VAR_GLOBAL
     g_xFirstPass: BOOL := TRUE;
    g_xIOState	:	BOOL := FALSE;
    g_aEcatMaster1 AT %I* : AMSNETID;
    g_aEcatMaster2 AT %I* : AMSNETID;
END_VAR

(* stored: Version 1.1.0.1, ProductVersion 3.1.4022.18
   GVL GVL: Id {f639b635-2ac5-4d16-9ee0-ff8224cf5b4c} *)
